FUNCTION_BLOCK FB_BAR (* An orientable single bar graph *)
  (* Standard: 61499-1 *)
  (* Version 0.3, 2004-08-20, JHC, Rockwell Automation, Corrected documentation of output. *)
  (* Version 0.2, 2004-01-20, JHC, Rockwell Automation, Corrected documentation of STYLE input. *)
  (* Version 0.1, 2000-04-28, JHC, Rockwell Automation, Added STYLE input *)
  (* Compiler header: package fb.rt.hmi; import java.awt.*; *)
  (* Compiler Java Sun JDK 1.3.1 *)
  (* Compiler Java IBM VisualAge 3.0 *)
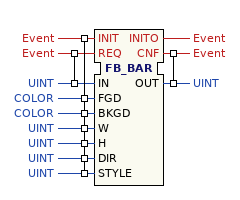
  EVENT_INPUT
    INIT WITH FGD, BKGD, W, H, DIR, STYLE; (* Initialization Request *)
    REQ WITH IN; (* Update the bar *)
  END_EVENT
  EVENT_OUTPUT
    INITO; (* Initialization Confirm *)
    CNF WITH OUT; (* REQ Confirmation *)
  END_EVENT
  VAR_INPUT
    IN : UINT; (* Value to display *)
    FGD : COLOR := red; (* Foreground Color *)
    BKGD : COLOR := blue; (* Background Color *)
    W : UINT; (* Bar width *)
    H : UINT; (* Bar height *)
    DIR : UINT; (* Orientation:0=L/R,1=T/B,2=R/L,3=B/T *)
    STYLE : UINT; (* Style:0=BAR,1=SLIDER *)
  END_VAR
  VAR_OUTPUT
    OUT : UINT; (* Displayed value,limited from 0% to 100% *)
  END_VAR
END_FUNCTION_BLOCK
